{attribute 'qualified_only'}


VAR_GLOBAL
    glv_a : bool;
END_VAR

(* stored: Version 1.1.0.1, ProductVersion 3.1.4024.16
   GVL GVL: Id {0bf22201-58db-4557-8ff8-481092298ecc} *)
